// Mitsubishi GX Works2 project: Flip-flop practice 2   PLC: Q03UDV

PROGRAM MAIN
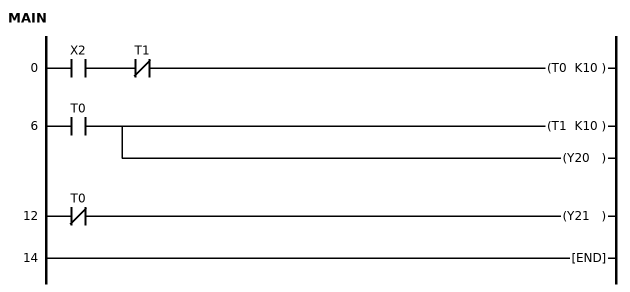
0     LD      X2
      ANI     T1
      OUT     T0 K10
6     LD      T0
      OUT     T1 K10
      OUT     Y20
12    LDI     T0
      OUT     Y21
14    END
END_PROGRAM
